FUNCTION_BLOCK ABSTRACT FB_Abstract


// This Function Block can't be instaniated but has to be extended.

METHOD PROTECTED M_Cycle : BOOL
VAR_INPUT
END_VAR

// This Method does not have to be incorporated into child class
END_METHOD

METHOD PROTECTED ABSTRACT M_Init : BOOL
VAR_INPUT
END_VAR


// This Method has to be incorporated into child class
END_METHOD

END_FUNCTION_BLOCK

(* stored: Version 1.1.0.1
   POU FB_Abstract: Id {27e5f71f-24af-4280-8f09-ea2bb114ab87}, SpecialFunc None
   Method M_Cycle: Id {3b8b170d-8710-47e0-a7fb-acf281279ebc}
   Method M_Init: Id {15d79c0a-047b-4eb5-b25d-e0e45f70083a} *)
